FUNCTION_BLOCK ReadRecipeFromFile
VAR_INPUT
END_VAR
VAR_OUTPUT
END_VAR
VAR
END_VAR

END_FUNCTION_BLOCK

(* stored: Version 1.1.0.1, ProductVersion 3.1.4022.18
   POU ReadRecipeFromFile: Id {f2ca5823-87be-4e5b-a7f8-ec8da86c7b10}, SpecialFunc None *)
